(* PLC project Unnamed, Unknown Unnamed 1 *)
(* stored: creationDateTime 2025-10-17T14:24:37, modificationDateTime 2025-10-17T14:34:49 *)

PROGRAM program0
  VAR
    Button : BOOL;
    Output : BOOL;
  END_VAR

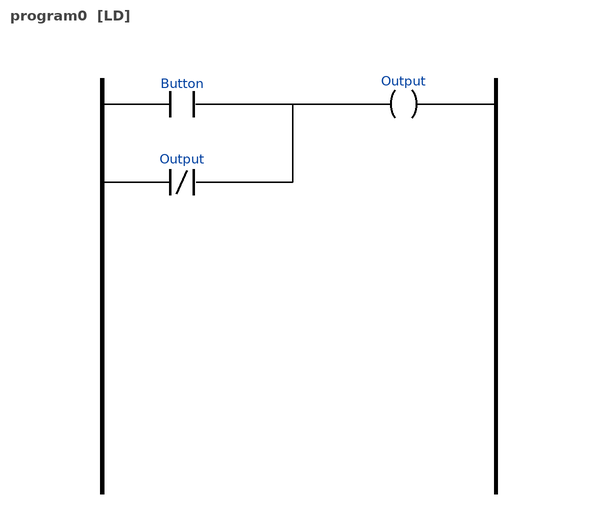
(* LD diagram, written out as Structured Text *)
Output := Button OR NOT Output;
END_PROGRAM

CONFIGURATION Config0
  RESOURCE Res0 ON PLC
    TASK task0(INTERVAL := T#20ms, PRIORITY := 0);
    PROGRAM instance0 WITH task0 : program0;
  END_RESOURCE
END_CONFIGURATION
